TYPE CmpCore :
STRUCT
	
	Framework: Framework;

END_STRUCT
END_TYPE

(* stored: Version 1.1.0.1, ProductVersion 3.1.4024.6
   DUT CmpCore: Id {6f9d3c06-3816-4efe-826b-369f5e76fcf4} *)
